// Annex I I.10.2 - one offset from the nest pose, in the nest's own frame.
TYPE ST_ApproachStep :
STRUCT
    D         : ST_RobotPose;   // offset applied to the nest pose
    MoveClass : E_MoveClass;
END_STRUCT
END_TYPE

(* stored: Version 1.1.0.1, ProductVersion 3.1.4024.12
   DUT ST_ApproachStep: Id {f6989268-9469-477d-a8c3-d8812a254c94} *)
